// TIA Portal V18 export
FUNCTION "AOProxy" : Void   // FC59001, LAD
{ S7_Optimized_Access := 'TRUE' }
VERSION : 0.1
// stored: AutoNumber false, IsIECCheckEnabled false, SetENOAutomatically false, UDAEnableTagReadback false
   VAR_INPUT
      iUnitID : Int;
      cCHModeCtrl : Byte;
      rDriverSignal : Real;
      rDrivenSignal : Real;
      xProxyIsOnInd : Bool;
      xProxyIsOffInd : Bool;
   END_VAR
   VAR_IN_OUT
      rProxySignal : Real;
      xProxyCmd : Bool;
      xProxyIndError : Bool;
   END_VAR
BEGIN

REGION Network 1 (SCL)
   CASE #cCHModeCtrl OF
       0:  // Not Active
           #xProxyCmd := FALSE;
           #rProxySignal := 0.0;
       1:  // Straignt signal
           #xProxyCmd := TRUE;
           #rProxySignal := #rDrivenSignal;
       2:  // Driven Initial signal
           #xProxyCmd := TRUE;
           #rProxySignal := #rDrivenSignal;
       3:  // Replace initial signal
           #xProxyCmd := TRUE;
           #rProxySignal := #rDriverSignal;
   END_CASE;
END_REGION
END_FUNCTION
